	4: (*wait for answer - upload*)
		TimeStart 							:= TRUE; 						// restart timer fot timeout (for each packet)
		// expect and save packet
		IF FML_REF.RespID = FML_FPC_RESP_file_done AND FML_REF.FPCS_Packet.Control = FML_REF.FPCC_Packet.Control AND FML_REF.FPCS_Packet.BitSequenceNr = Sequence THEN
			Buffer							:= FML_REF.FPCS_Packet.Data;	// write incoming data from controller into buffer (6 Byte)
			FOR i := 0 TO 5 DO
				PtrToDataFileArray^			:= Buffer[i+1];					// write data from buffer to output (each byte separately)
				PtrToDataFileArray			:= PtrToDataFileArray + 1;
			END_FOR
			
			CountByte 						:= CountByte + udLength;		// count up the bytes
			NextSequence();       											// count sequence
			TimeStart						:= FALSE;
			Step							:= 3; 
		
		// finish upload, controller sends stopp
		ELSIF FML_REF.RespID = FML_FPC_RESP_file_done AND FML_REF.FPCS_Packet.Control = FML_FPC_FILE_TRANSFER_stop AND FML_REF.FPCS_Packet.BitSequenceNr = Sequence THEN
			TimeStart 						:= FALSE;
			IF CountByte <> Filesize OR CountByte < 100 THEN 				// check if all bytes are uploaded
				Step 			    		:= 21; 							// wrong size --> error state
				Status.Err:=TRUE; Status.Cat:=FML_parameter_transfer; Status.ID:=FML_incomplete; 
			ELSE
				Step 			    		:= 20;							// size is right, upload successful, end state		
			END_IF
						
		// error from controller, general EFPC error
		ELSIF FML_REF.RespID = FML_FPC_RESP_error THEN
			Status.Err:=TRUE; Status.Cat:=FML_parameter_transfer; Status.ID:=FML_REF.FPCS_Packet.Data[1]+1000; 
			TimeStart 						:= FALSE;
			NextSequence();     											// count sequence modul
			Step 			  				:= 23;  						// send stopp after error
			
		// error from controller - upload
		ELSIF FML_REF.FPCS_Packet.Control = FML_FPC_FILE_TRANSFER_error THEN
			Status.Err:=TRUE; Status.Cat:=FML_parameter_transfer; Status.ID:=FML_REF.FPCS_Packet.Data[1]+1000; 	// get error code from data at byte 1
			TimeStart						:= FALSE;
			NextSequence();     											// count sequence modulo
			Step							:= 23;  						// send stopp after error	
		
		ELSE 
			//timeout
			IF TimeStop THEN
				Status.Err:=TRUE; Status.Cat:=FML_parameter_transfer; Status.ID:=FML_time_out; 
				Step						:= 21;  						// send error message to controller
				TimeStart					:= FALSE;
			END_IF	
		END_IF
	
	6: (*start requirement - download*)
		FOR i := 0 TO 5 DO
			Buffer[i+1]						:= PtrToDataFileArray^;			// write data from data array (input) into buffer (each byte separately)
			PtrToDataFileArray				:= PtrToDataFileArray + 1;
		END_FOR

		IF Sequence = 0 THEN    											
			CalculateFilesize(); 											// calculate size of file as a multiple of udLength
			
			IF FileSize < 262 THEN  										// file larger than header --> error
				Step 						:= 27;
				Status.Err:=TRUE; Status.Cat:=FML_parameter_transfer; Status.ID:=FML_size_err; 
				RETURN;
			ELSIF FileSize > SizeOfFileArray THEN							// check if the array is big enough
				Step 			    		:= 27; 							// array is to small --> error state
				Status.Err:=TRUE; Status.Cat:=FML_parameter_transfer; Status.ID:=FML_volume_err;
				RETURN;
			END_IF
		END_IF	
				
		FML_REF.FPCC_Packet.Data 			:= Buffer;						// write data from buffer to controller (6 byte)	
		CountByte 							:= CountByte + udLength;
		FML_REF.FPCC_Modus					:= 4;							// modus parameter file 
		FML_REF.ReqID						:= FML_FPC_REQ_write_file; 		// download
		FML_REF.FPCC_Packet.Control			:= FML_FPC_FILE_TRANSFER_start; // start transfer
		FML_REF.FPCC_Packet.BitSequenceNr	:= Sequence;
		TimeStart 							:= TRUE;
		Step 								:= 7;

			
	7: (*wait for response from controller - download*)
		IF FML_REF.RespID = FML_FPC_RESP_file_done AND FML_REF.FPCS_Packet.Control = FML_REF.FPCC_Packet.Control AND FML_REF.FPCS_Packet.BitSequenceNr = Sequence THEN
			Sequence 						:= 1;
			Step 							:= 8;
		ELSE
			//timeout
			IF TimeStop THEN
				TimeStart 					:= FALSE;
				Step 						:= 9;
			END_IF
		END_IF

	8: (*send packet - download*)
		IF CountByte < FileSize THEN
			FOR i := 0 TO 5 DO
				Buffer[i+1]					:= PtrToDataFileArray^;			// write data from data array (input) into buffer (each byte separately)
			PtrToDataFileArray				:= PtrToDataFileArray + 1;
		END_FOR
		
		FML_REF.FPCC_Packet.Data 				:= Buffer;					// write data from buffer to controller (6 byte)
			CountByte							:= CountByte + udLength;
			FML_REF.FPCC_Packet.Control			:= FML_FPC_FILE_TRANSFER_active;
			FML_REF.FPCC_Packet.BitSequenceNr	:= Sequence;
			Step								:= 9;
				
		ELSE          //---- end of file detected -ä stop to device
			FML_REF.FPCC_Packet.Control 		:= FML_FPC_FILE_TRANSFER_stop;
			FML_REF.FPCC_Packet.BitSequenceNr	:= Sequence;
			FML_REF.FPCC_Packet.Data 			:= Buffer;
			Step								:= 9;
		END_IF
	
	9: (*wait for confirmation of receipt of controller - download*)
		// receive and process message 
		TimeStart								:= TRUE;
		IF FML_REF.RespID = FML_FPC_RESP_file_done AND FML_REF.FPCS_Packet.Control = FML_FPC_FILE_TRANSFER_active AND FML_REF.FPCS_Packet.BitSequenceNr = Sequence THEN
			NextSequence();														// count sequence modulo
			TimeStart							:= FALSE;       												
			Step								:= 8;
			
		// if stop has been sent to the controller
		ELSIF FML_REF.RespID = FML_FPC_RESP_file_done AND FML_REF.FPCS_Packet.Control = FML_FPC_FILE_TRANSFER_stop AND FML_REF.FPCS_Packet.BitSequenceNr = Sequence THEN
			IF CountByte <> Filesize OR CountByte < 100 THEN 					// check if parameterfile has been loaded
				Step 			:= 21; 											// wrong size, error step
				Status.Err:=TRUE; Status.Cat:=FML_parameter_transfer; Status.ID:=FML_incomplete;
			ELSE
				Step 			:= 20;											// right size, download successful, end state    // check if all bytes are uploaded
			END_IF
			TimeStart 			:= FALSE;
			
		// error from controller, general EFPC error
		ELSIF FML_REF.RespID = FML_FPC_RESP_error THEN
			Status.Err:=TRUE; Status.Cat:=FML_parameter_transfer; Status.ID:=FML_REF.FPCS_Packet.Data[1]+1000;	// get error code from data at byte 1
			NextSequence();       												// count sequence modulo
			Step				:= 23;
			TimeStart 			:= FALSE;
			
		// error form controller - Download
		ELSIF FML_REF.FPCS_Packet.Control = FML_FPC_FILE_TRANSFER_error THEN
			Status.Err:=TRUE; Status.Cat:=FML_parameter_transfer; Status.ID:=FML_REF.FPCS_Packet.Data[1]+1000;	// get error code from data at byte 1
      		NextSequence();       												// count sequence modulo
			IF Status.ID = FML_par_file_err THEN								// If Status.ID == 1008
				Step 			:= 27;
			ELSE
				Step 			:= 23;
			END_IF
			TimeStart 			:= FALSE;
		
		ELSE
			// timeout
			IF TimeStop THEN
				Status.Err:=TRUE; Status.Cat:=FML_parameter_transfer; Status.ID:=FML_time_out; 
				Step 			:= 21;
				TimeStart		:= FALSE;
			END_IF
		END_IF
	
	20:	(*  ==== done with no error ==== *)
		Status.Err:=FALSE; Status.Cat:=FML_no_category; Status.ID:=FML_no_error;
		Step					:= 27;      						// wait for NOT execute
	
		
	21: (*send error message to Controller*)
		NextSequence();      				 						// count sequence modulo
		FML_REF.FPCC_Modus 					:= 4;
		FML_REF.FPCC_Packet.Control 		:= 3;
		FML_REF.FPCC_Packet.BitSequenceNr  	:= Sequence;
		FML_REF.FPCC_Packet.Data 			:= Buffer;
		TimeStart							:= TRUE;
		Step 								:= 22;
			
	22: (*wait for error message from controller*)
		IF FML_REF.RespID = FML_FPC_RESP_file_done AND FML_REF.FPCS_Packet.Control = FML_FPC_FILE_TRANSFER_error THEN
			NextSequence();       									// count sequence modulo
			TimeStart						:= FALSE;
			Step 							:= 23;
		ELSE
			IF TimeStop THEN
				Status.Err:=TRUE; Status.Cat:=FML_parameter_transfer; Status.ID:=FML_time_out;
				TimeStart 					:= FALSE;
				Step 						:= 23;
			END_IF
		END_IF
		
	23: (*send STOPP after error*)	
		FML_REF.FPCC_Packet.Control 		:= 2; 					// after error STOPP is sending to Controller
		FML_REF.FPCC_Packet.BitSequenceNr 	:= Sequence;
		FML_REF.FPCC_Packet.Data 			:= Buffer;
		TimeStart 							:= TRUE;
		Step 								:= 24;		
		
	24: (*query wheater stop was confirmed by controller*)
		IF (FML_REF.RespID = FML_FPC_RESP_file_done AND FML_REF.FPCS_Packet.Control = 2) OR  FML_REF.RespID = 7 THEN
			Step 							:= 27;
			TimeStart 						:= FALSE;
		ELSIF FML_REF.RespID = FML_FPC_RESP_file_done AND FML_REF.FPCS_Packet.Control = 3 AND SendRepeat < 4 THEN
			Status.ID						:= FML_REF.FPCS_Packet.Data[1]+1000;			// get error code from data at byte 1
			IF Status.ID <> 1000 THEN
				Status.Err					:= TRUE;
				Status.Cat					:= FML_parameter_transfer;
			END_IF
			
			Sequence 						:= Sequence + 1;
			SendRepeat 						:= SendRepeat + 1;
			TimeStart 						:= FALSE;
			Step 							:= 23;
		ELSE
			// timeout
			IF TimeStop THEN
				Status.Err:=TRUE; Status.Cat:=FML_parameter_transfer; Status.ID:=FML_time_out;
				TimeStart 					:= FALSE;
				Step 						:= 27;
			END_IF
		END_IF
		
  
  27: (*idle - wait for execute = false*)
		vis_upload 							:= FALSE;
		vis_download 						:= FALSE;
		Done								:= TRUE;
		Step								:= 30;
    		
  30: (*do nothing - wait for NOT execute*)
    	;
  
END_CASE

Status.Msg				:= GetStatusMessage(Status);
Error					:= Status.Err;

(* ===== end of function block ============================= *)

ACTION CalculateFilesize:
(* -----------------------------------------------------
   This action calculates the file size as a couple of 6 
   from the first 2 bytes of the buffer
   ----------------------------------------------------- *)

 	FileSize	:= DWORD_TO_DINT( SHL(BYTE_TO_DWORD(pbyBuffer^[2]),8) OR pbyBuffer^[1]); 	// length of data field
	FileSize	:= (Filesize + 2 * udLength -1) / udLength ; 								// +6: size of parameter file at first position, +5 und /6 for rounding up 
	FileSize	:= FileSize * udLength; 													// bytesize is being computed out of number of packages
END_ACTION

ACTION NextSequence:
(* -----------------------------------------------------
   This action increments the Sequence counter modulo 32. 
   It is used at 8 points in CMMO_ST_PRM_FILE
   ----------------------------------------------------- *)
	IF Sequence = 31 THEN
		Sequence 	:= 0;
	ELSE
		Sequence 	:= Sequence + 1;
	END_IF
END_ACTION

END_FUNCTION_BLOCK

// Blocks/Parameterize/FPC_DIRMP
(* ============================================================================
   FESTO AG & Co. KG, Esslingen - Copyright 2015. All rights reserved.                       
 ------------------------------------------------------------------------------
 Functionblock:  PRM_DIRMP  
 Description:    function block to pass dynamic parameter values for direct-mode-positioncontrol
 Version:        V3.5.7.21        
 Composer:       bejk
 Last update:    13.11.2017                                                                           
------------------------------------------------------------------------------- *)
{library private}
(* -----------------------------------------------------------------------------
Date        Name            	Activity                                                                              
11.03.2009  Benjamin Kilgus 	created
            Rudolf Schenke  	PNU array created 
09.02.2015  Rudolf Schenke  	Implement 16-bit mode with hide preset 
22.06.2015	Christian Hammer	adaptation to use this FB for all drives
04.09.2015  Christian Hammer	error handling (deleted RETVAL, created Status)
13.11.2017	Christian Hammer	added blockade of FB for SFC-DC and MTR-DCI controller
=============================================================================== *)
{library public}

(* use this function block only with the function blocks FML_Read and FML_Write *)

FUNCTION_BLOCK FPC_DIRMP

VAR_IN_OUT
	FML_REF					: DT_FML_REF;		// structure of the parameter to control and parametrize the motorcontroller
END_VAR

VAR_INPUT
	Execute             	: BOOL;				// perfrom data exchange
	Write               	: BOOL;				// read or write the parameter	(1=write/0=read)
	Velocity            	: DINT;				// base velocity directmode positioning
	Acceleration			: DINT; 			// acceleration directmode positioning
 	Deceleration        	: DINT; 			// deceleration directmode positioning
END_VAR

VAR_OUTPUT	
	Done                	: BOOL;				// transmission done
	Error					: BOOL; 			// transmission fault
	Status					: DT_FML_STATUS;	// structure with the status information of the function block and FPC
	ActVelocity         	: DINT;  			// base velocity directmode positioning
	ActAcceleration     	: DINT;  			// acceleration directmode positioning
	ActDeceleration     	: DINT;  			// deceleration directmode positioning
END_VAR

{library private}
VAR
	bInit           		: BOOL	:=FALSE;										// status of inizialisation of the FB
	lMemberID   			: INT;													// local member ID of the FB													
	Param       			: ARRAY [1..maxParamCount] OF DT_FML_PRM_DESCRIPTION;	// parameter to write in motorcontroller
	listPNU    				: ARRAY [1..maxParamCount] OF INT := [540,541,542];		// PNUs for the parameter 
	Step        			: INT:= 0; 												// actual step number 
	ixPar       			: INT:= 1;  											// index for the array

	TONInst					: TON;													// timer instance to monitor a timeout of the function block
	TimeStart				: BOOL;													// variable to start the timer instance
	TimeoutTime				: TIME := T#3S;											// timeout time 	
END_VAR

VAR CONSTANT
	maxParamCount			: INT := 3;												// max number of the parameter 
END_VAR

{library public}

(* ====== initial block routine ===================================== *)
(* ----- get MemberID for this function block ------------------------*)
IF NOT bInit THEN
	FML_REF.MemberIDmax		:= FML_REF.MemberIDmax +1;
	lMemberID				:= FML_REF.MemberIDmax;
	bInit					:= TRUE;
	Status.Err:=FALSE; Status.Cat:=FML_function_block; Status.ID:=FML_init_active;
END_IF


(* ====== supervision of timeout ==================================== *)
(* ----- timer to monitor a timeout of the function block ------------*)
TONInst(IN := TimeStart, PT := TimeoutTime);
IF TONInst.Q THEN
	Status.Err:=TRUE; Status.Cat:=FML_function_block; Status.ID:=FML_fb_timeout;
	Done					:= TRUE;
	Step					:= 30;
END_IF

// this function block is not usable with SFC-DC and MTR-DCI
IF Execute 
	AND	((FML_REF.DeviceType = SFC_DC)
	OR (FML_REF.DeviceType = MTR_DCI)) THEN
		Done				:= TRUE;
		Status.Err:=TRUE; Status.Cat:=FML_function_block; Status.ID:=FML_wrong_device;
		Step				:= 100;
END_IF

IF Param[1].PNU = 0 THEN
  FOR ixPar:=1 TO maxParamCount DO
    Param[ixPar].PNU 		:= listPNU[ixPar]; 			// fill in the PNU
    Param[ixPar].SUBINDEX 	:= 1;         				// fill in a fix subindex
	END_FOR
    // 1 =  540.1: Paramter Direktbetrieb Basisgeschwindigkeit directmode positioning
    // 2 =  541.1: Paramter Beschleunigung directmode positioning
    // 3 =  542.1: Paramter Verzögerung directmode positioning
END_IF;

(* ===== logic part ================================================= *)
IF NOT Execute AND (Step <> 0) THEN   					// aborting FB
	FML_REF.MemberID		:= 0;
	FML_REF.ReqID        	:= FML_FPC_REQ_none;
	FML_REF.PNU       		:= 0;
	FML_REF.Subindex   		:= 0;
	FML_REF.Value			:= 0;
	ActVelocity				:= 0;
	ActAcceleration			:= 0;
	ActDeceleration			:= 0;
 	Step                    := 0;
END_IF

CASE Step OF
  0:(* *)
  Done						:= FALSE;
  TimeStart					:= FALSE;
  Status.Err:=FALSE; Status.Cat:=FML_no_category; Status.ID:=FML_no_error;

	IF (FML_REF.MemberID = 0) AND Execute THEN 	
		Status.Err:=FALSE; Status.Cat:=FML_function_block; Status.ID:=FML_fb_busy;
		
		IF (FML_REF.DeviceType = CMMP_AS) 
		OR (FML_REF.DeviceType = CMMS_AS) 
		OR (FML_REF.DeviceType = CMMS_ST)
		OR (FML_REF.DeviceType = CMMD_AS) THEN					(* CMMP-AS or CMMS_AS or CMMS_ST or CMMD_AS *)	
			FML_REF.FPCC_Modus 	:= E_FML_FPC_MODUS.FML_FPC_MODUS_PNU_11BIT;
		ELSE 												(*******EMCA-EC or CMMO-ST*******)	
			FML_REF.FPCC_Modus 	:= E_FML_FPC_MODUS.FML_FPC_MODUS_PNU_16BIT;
		END_IF
    	FML_REF.MemberID		:= lMemberID;
		FML_REF.ReqID			:= FML_FPC_REQ_none;
		FML_REF.PNU				:= 0;
		FML_REF.Subindex		:= 0;
		FML_REF.Value			:= 0;
		ixPar					:= 1;  						// set to 1st array element
		(* writing *)
		IF Write THEN
			Param[1].Value		:= Velocity;
			Param[2].Value		:= Acceleration;
			Param[3].Value		:= Deceleration;
			Step				:= 10;
		(* reading *)
		ELSE
			Step				:= 20;
		END_IF
	ELSIF (FML_REF.MemberID <> lMemberId) AND Execute THEN
		Status.Err:=FALSE; Status.Cat:=FML_function_block; Status.ID:=FML_other_fb_active;
	END_IF

  10:(* writing parameter[ixPar] *)
  	TimeStart					:= TRUE;
	IF NOT FML_REF.Done THEN
		TimeStart				:= FALSE;  
		FML_REF.ReqID			:= FML_FPC_REQ_write_array_dword;
		FML_REF.PNU				:= Param[ixPar].PNU;
		FML_REF.Subindex		:= Param[ixPar].SUBINDEX;
		FML_REF.Value			:= Param[ixPar].VALUE;
		Step					:= 11;
	END_IF

  11:(* *)
  	TimeStart					:= TRUE;
	IF FML_REF.Done AND NOT FML_REF.Err THEN
		TimeStart				:= FALSE;
		FML_REF.ReqID			:= FML_FPC_REQ_none;
		ixPar					:= ixPar +1;
		Step					:= 10;
		IF ixPar > maxParamCount THEN
		  	Done					:= TRUE;
		  	ActVelocity			:= Param[1].VALUE;
			ActAcceleration		:= Param[2].VALUE;
			ActDeceleration		:= Param[3].VALUE;
		  	Status.Err:=FALSE; Status.Cat:=FML_no_category; Status.ID:=FML_no_error;
		  	Step				:= 30;
		END_IF
	ELSIF FML_REF.Done AND FML_REF.Err THEN
		TimeStart				:= FALSE; 
		Done					:= TRUE;
		Status.Err:=TRUE; Status.Cat:=FML_parameter_transfer; Status.ID:=FML_REF.ActValue;
		Step					:= 30;
	END_IF

  20: (* reading *)
  	TimeStart					:= TRUE;
	IF NOT FML_REF.Done THEN
		TimeStart				:= FALSE;
		FML_REF.ReqID			:= FML_FPC_REQ_read_array;
 		FML_REF.PNU				:= Param[ixPar].PNU;
 		FML_REF.Subindex		:= Param[ixPar].SUBINDEX;
 		Step					:= 21;
	END_IF

  21:(* set ouput variables*)
  	TimeStart					:= TRUE;
	IF FML_REF.Done AND NOT FML_REF.Err THEN
		TimeStart				:= FALSE;  
		FML_REF.ReqID			:= FML_FPC_REQ_none;
		Param[ixPar].Value		:= FML_REF.ActValue;
		ixPar					:= ixPar +1;
		Step					:= 20;
		IF ixPar > maxParamCount THEN
			ActVelocity			:= Param[1].VALUE;
			ActAcceleration		:= Param[2].VALUE;
			ActDeceleration		:= Param[3].VALUE;
			Done				:= TRUE;
			Status.Err:=FALSE; Status.Cat:=FML_no_category; Status.ID:=FML_no_error;
			Step				:= 30;
		END_IF
	ELSIF FML_REF.Done AND FML_REF.Err THEN
		TimeStart				:= FALSE;  
		Done					:= TRUE;
		Status.Err:=TRUE; Status.Cat:=FML_parameter_transfer; Status.ID:=FML_REF.ActValue;
		Step					:= 30;
	END_IF

  30: (* done - do nothing *)
	  ;
	  
END_CASE;

Status.Msg				:= GetStatusMessage(Status);
Error					:= Status.Err;

(* ===== end of function block ============================= *)

END_FUNCTION_BLOCK

// VISU/VIS_FPC_PNU
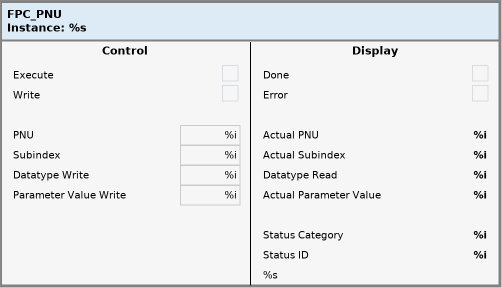
VISUALIZATION VIS_FPC_PNU  // 502x288
VAR_INPUT
	{attribute 'parameterstringof' := 'm_Input_INST'}
	m_Input_INST_Str 	: STRING;
END_VAR
VAR_IN_OUT
	m_Input_INST 		: FPC_PNU;
END_VAR
    Rectangle (0,1 500x285)
    Rectangle (0,1 500x40), "FPC_PNU Instance: %s", text variable: m_Input_INST_Str
    Rectangle (260,265 240x20), "%s", text variable: m_Input_INST.Status.Msg
    Rectangle (180,125 60x20), "%i", text variable: m_Input_INST.PNU
        OnMouseDown: write the text variable via Edit
    Rectangle (180,165 60x20), "%i", text variable: m_Input_INST.DatatypeWR
        OnMouseDown: write the text variable via Edit
    Rectangle (430,125 60x20), "%i", text variable: m_Input_INST.ActPNU
    Label (10,65 120x20), "Execute"
    Label (10,85 120x20), "Write"
    RoundedRectangle (222,65 16x16), colour toggle: m_Input_INST.Execute
        toggle m_Input_INST.Execute
    RoundedRectangle (222,85 16x16), colour toggle: m_Input_INST.Write
        toggle m_Input_INST.Write
    Label (10,125 120x20), "PNU"
    Label (10,165 120x20), "Datatype Write"
    Label (260,65 120x20), "Done"
    Label (260,85 120x20), "Error"
    RoundedRectangle (472,65 16x16), colour toggle: m_Input_INST.Done
    RoundedRectangle (472,85 16x16), colour toggle: m_Input_INST.Error
    Label (260,125 128x20), "Actual PNU"
    Label (0,41 250x20), "Control"
    Label (250,41 250x20), "Display"
    Line (250,42) (250,285)
    Rectangle (430,165 60x20), "%i", text variable: m_Input_INST.DatatypeRD
    Label (260,165 128x20), "Datatype Read"
    Rectangle (180,145 60x20), "%i", text variable: m_Input_INST.Subindex
        OnMouseDown: write the text variable via Edit
    Rectangle (430,145 60x20), "%i", text variable: m_Input_INST.ActSubindex
    Label (10,145 120x20), "Subindex"
    Label (260,145 128x20), "Actual Subindex"
    Rectangle (430,225 60x20), "%i", text variable: m_Input_INST.Status.Cat
    Label (260,225 128x20), "Status Category"
    Rectangle (430,245 60x20), "%i", text variable: m_Input_INST.Status.ID
    Label (260,245 128x20), "Status ID"
    Rectangle (180,185 60x20), "%i", text variable: m_Input_INST.Value
        OnMouseDown: write the text variable via Edit
    Label (10,185 120x20), "Parameter Value Write"
    Rectangle (430,185 60x20), "%i", text variable: m_Input_INST.ActValue
    Label (260,185 128x20), "Actual Parameter Value"
END_VISUALIZATION

// VISU/VIS_FPC_DIAG_BUFFER
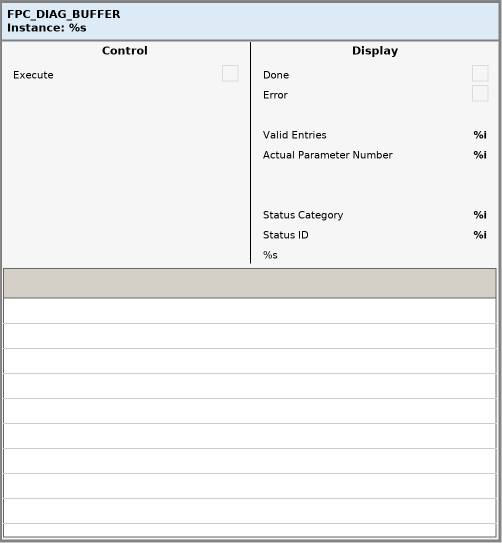
VISUALIZATION VIS_FPC_DIAG_BUFFER  // 502x543
VAR_INPUT
	{attribute 'parameterstringof' := 'm_Input_INST'}
	m_Input_INST_Str 	: STRING;
END_VAR
VAR_IN_OUT
	m_Input_INST 		: FPC_DIAG_BUFFER;
END_VAR
    Rectangle (0,1 500x540)
    Rectangle (0,1 500x40), "FPC_DIAG_BUFFER Instance: %s", text variable: m_Input_INST_Str
    Rectangle (260,245 240x20), "%s", text variable: m_Input_INST.Status.Msg
    Rectangle (430,145 60x20), "%i", text variable: m_Input_INST.ParamNo
    Label (10,65 120x20), "Execute"
    RoundedRectangle (222,65 16x16), colour toggle: m_Input_INST.Execute
        toggle m_Input_INST.Execute
    Label (260,65 120x20), "Done"
    Label (260,85 120x20), "Error"
    RoundedRectangle (472,65 16x16), colour toggle: m_Input_INST.Done
    RoundedRectangle (472,85 16x16), colour toggle: m_Input_INST.Error
    Label (260,145 140x20), "Actual Parameter Number"
    Label (0,41 250x20), "Control"
    Label (250,41 250x20), "Display"
    Line (250,42) (250,263)
    Rectangle (430,205 60x20), "%i", text variable: m_Input_INST.Status.Cat
    Label (260,205 128x20), "Status Category"
    Rectangle (430,225 60x20), "%i", text variable: m_Input_INST.Status.ID
    Label (260,225 128x20), "Status ID"
    Rectangle (430,125 60x20), "%i", text variable: m_Input_INST.ValidEntries
    Label (260,125 140x20), "Valid Entries"
    Table (3,268 493x269), data array: m_Input_INST.astVisu
        p3854506369: m_Input_INST.astVisu[INDEX].sEvent
        p1892666644: m_Input_INST.astVisu[INDEX].sStamp
        p338671338: m_Input_INST.astVisu[INDEX].sFault
        p2170511999: m_Input_INST.astVisu[INDEX].sText
        p511219082: TimeStamp
        p1755163831: Message #
        p4092479075: Message Description
END_VISUALIZATION

// VISU/VIS_FPC_DIRMP
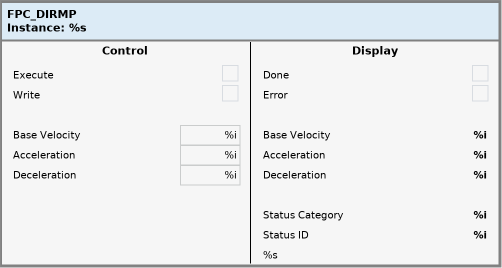
VISUALIZATION VIS_FPC_DIRMP  // 502x268
VAR_INPUT
	{attribute 'parameterstringof' := 'm_Input_INST'}
	m_Input_INST_Str 	: STRING;
END_VAR
VAR_IN_OUT
	m_Input_INST 		: FPC_DIRMP;
END_VAR
    Rectangle (0,1 500x265)
    Rectangle (0,1 500x40), "FPC_DIRMP Instance: %s", text variable: m_Input_INST_Str
    Rectangle (260,245 240x20), "%s", text variable: m_Input_INST.Status.Msg
    Rectangle (180,125 60x20), "%i", text variable: m_Input_INST.Velocity
        OnMouseDown: write the text variable via Edit
    Rectangle (180,165 60x20), "%i", text variable: m_Input_INST.Deceleration
        OnMouseDown: write the text variable via Edit
    Rectangle (430,125 60x20), "%i", text variable: m_Input_INST.ActVelocity
    Label (10,65 120x20), "Execute"
    Label (10,85 120x20), "Write"
    RoundedRectangle (222,65 16x16), colour toggle: m_Input_INST.Execute
        toggle m_Input_INST.Execute
    RoundedRectangle (222,85 16x16), colour toggle: m_Input_INST.Write
        toggle m_Input_INST.Write
    Label (10,125 120x20), "Base Velocity"
    Label (10,165 120x20), "Deceleration"
    Label (260,65 120x20), "Done"
    Label (260,85 120x20), "Error"
    RoundedRectangle (472,65 16x16), colour toggle: m_Input_INST.Done
    RoundedRectangle (472,85 16x16), colour toggle: m_Input_INST.Error
    Label (260,125 128x20), "Base Velocity"
    Label (0,41 250x20), "Control"
    Label (250,41 250x20), "Display"
    Line (250,42) (250,263)
    Rectangle (430,165 60x20), "%i", text variable: m_Input_INST.ActDeceleration
    Label (260,165 128x20), "Deceleration"
    Rectangle (180,145 60x20), "%i", text variable: m_Input_INST.Acceleration
        OnMouseDown: write the text variable via Edit
    Rectangle (430,145 60x20), "%i", text variable: m_Input_INST.ActAcceleration
    Label (10,145 120x20), "Acceleration"
    Label (260,145 128x20), "Acceleration"
    Rectangle (430,205 60x20), "%i", text variable: m_Input_INST.Status.Cat
    Label (260,205 128x20), "Status Category"
    Rectangle (430,225 60x20), "%i", text variable: m_Input_INST.Status.ID
    Label (260,225 128x20), "Status ID"
END_VISUALIZATION

// VISU/VIS_FPC_DATA_OBJECT
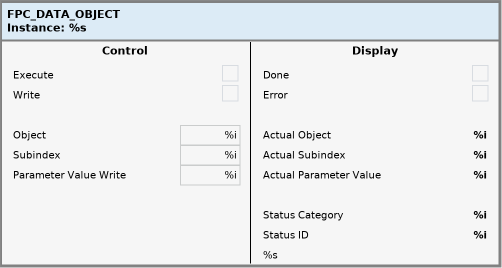
VISUALIZATION VIS_FPC_DATA_OBJECT  // 502x268
VAR_INPUT
	{attribute 'parameterstringof' := 'm_Input_INST'}
	m_Input_INST_Str	: STRING;
END_VAR
VAR_IN_OUT
	m_Input_INST 		: FPC_DATA_OBJECT;
END_VAR
    Rectangle (0,1 500x265)
    Rectangle (0,1 500x40), "FPC_DATA_OBJECT Instance: %s", text variable: m_Input_INST_Str
    Rectangle (260,245 240x20), "%s", text variable: m_Input_INST.Status.Msg
    Rectangle (180,125 60x20), "%i", text variable: m_Input_INST.Object
        OnMouseDown: write the text variable via Edit
    Rectangle (180,165 60x20), "%i", text variable: m_Input_INST.Value
        OnMouseDown: write the text variable via Edit
    Rectangle (430,125 60x20), "%i", text variable: m_Input_INST.ActObject
    Label (10,65 120x20), "Execute"
    Label (10,85 120x20), "Write"
    RoundedRectangle (222,65 16x16), colour toggle: m_Input_INST.Execute
        toggle m_Input_INST.Execute
    RoundedRectangle (222,85 16x16), colour toggle: m_Input_INST.Write
        toggle m_Input_INST.Write
    Label (10,125 120x20), "Object"
    Label (10,165 120x20), "Parameter Value Write"
    Label (260,65 120x20), "Done"
    Label (260,85 120x20), "Error"
    RoundedRectangle (472,65 16x16), colour toggle: m_Input_INST.Done
    RoundedRectangle (472,85 16x16), colour toggle: m_Input_INST.Error
    Label (260,125 128x20), "Actual Object"
    Label (0,41 250x20), "Control"
    Label (250,41 250x20), "Display"
    Line (250,42) (250,263)
    Rectangle (430,165 60x20), "%i", text variable: m_Input_INST.ActValue
    Label (260,165 128x20), "Actual Parameter Value"
    Rectangle (180,145 60x20), "%i", text variable: m_Input_INST.Subindex
        OnMouseDown: write the text variable via Edit
    Rectangle (430,145 60x20), "%i", text variable: m_Input_INST.ActSubindex
    Label (10,145 120x20), "Subindex"
    Label (260,145 128x20), "Actual Subindex"
    Rectangle (430,205 60x20), "%i", text variable: m_Input_INST.Status.Cat
    Label (260,205 128x20), "Status Category"
    Rectangle (430,225 60x20), "%i", text variable: m_Input_INST.Status.ID
    Label (260,225 128x20), "Status ID"
END_VISUALIZATION

// VISU/VIS_FHPP_CTRL
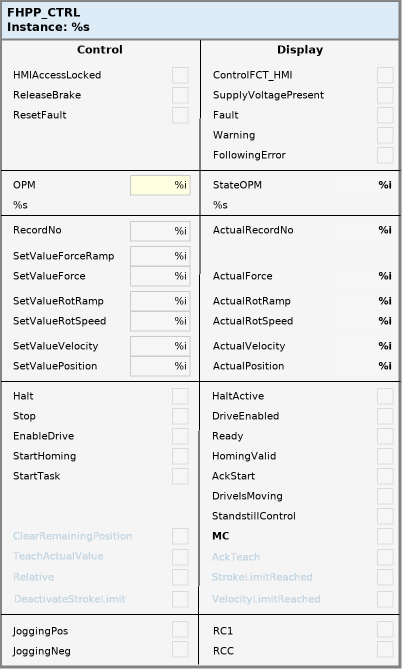
VISUALIZATION VIS_FHPP_CTRL  // 402x669
VAR_INPUT
	{attribute 'parameterstringof' := 'm_Input_INST'}
	m_Input_INST_Str 	: STRING;
END_VAR
VAR_IN_OUT
	m_Input_INST 		: FHPP_CTRL;
END_VAR
    Rectangle (0,1 400x666)
    Rectangle (0,0 400x40), "FHPP_CTRL Instance: %s", text variable: m_Input_INST_Str
    Rectangle (10,195 180x20), "%s", text variable: m_Input_INST.OPMString
    Rectangle (130,266 60x20), "%i", text variable: m_Input_INST.SetValueForce, colour toggle: (m_Input_INST.OPM) = 5
        OnMouseDown: write the text variable via Edit
    Rectangle (330,175 65x20), "%i", text variable: m_Input_INST.StateOPM
    Rectangle (130,336 60x20), "%i", tooltip "permissible range of value is 0 to 100", text variable: m_Input_INST.SetValueVelocity, colour toggle: (m_Input_INST.OPM= 1) or ((m_Input_INST.OPM =5) AND (m_Input_INST.tempVisuMode =2))
        OnMouseDown: write the text variable via Edit
    Rectangle (335,336 60x20), "%i", text variable: m_Input_INST.ActualVelocity, colour toggle: (m_Input_INST.StateOPM) = 1
    Rectangle (130,291 60x20), "%i", tooltip "permissible range of value is 0 to 100", text variable: m_Input_INST.SetValueRotRamp, colour toggle: m_Input_INST.OPM = 9
        OnMouseDown: write the text variable via Edit
    Rectangle (335,291 60x20), "%i", text variable: m_Input_INST.ActualRotRamp, colour toggle: (m_Input_INST.StateOPM) = 9
    Rectangle (130,311 60x20), "%i", text variable: m_Input_INST.SetValueRotSpeed, colour toggle: (m_Input_INST.OPM) = 9
        OnMouseDown: write the text variable via Edit
    Rectangle (335,311 60x20), "%i", text variable: m_Input_INST.ActualRotSpeed, colour toggle: (m_Input_INST.StateOPM) = 9
    Rectangle (130,356 60x20), "%i", text variable: m_Input_INST.SetValuePosition, colour toggle: (m_Input_INST.OPM) = 1
        OnMouseDown: write the text variable via Edit
    Rectangle (335,356 60x20), "%i", text variable: m_Input_INST.ActualPosition, colour toggle: (m_Input_INST.StateOPM = 1) or (m_Input_INST.StateOPM = 5) or (m_Input_INST.StateOPM = 0)
    Rectangle (210,195 180x20), "%s", text variable: m_Input_INST.StateOPMString
    Rectangle (335,266 60x20), "%i", text variable: m_Input_INST.ActualForce, colour toggle: (m_Input_INST.StateOPM) = 5
    Rectangle (335,220 60x20), "%i", text variable: m_Input_INST.ActualRecordNo, colour toggle: (m_Input_INST.StateOPM) = 0
    RoundedRectangle (377,428 16x16), colour toggle: m_Input_Inst.Ready
    RoundedRectangle (172,428 16x16), colour toggle: m_Input_Inst.EnableDrive
        toggle m_Input_Inst.EnableDrive
    RoundedRectangle (172,388 16x16), colour toggle: m_Input_Inst.Halt
        toggle m_Input_Inst.Halt
    RoundedRectangle (172,408 16x16), colour toggle: m_Input_Inst.Stop
        toggle m_Input_Inst.Stop
    RoundedRectangle (377,388 16x16), colour toggle: m_Input_Inst.HaltActive
    RoundedRectangle (377,408 16x16), colour toggle: m_Input_Inst.DriveEnabled
    RoundedRectangle (172,448 16x16), colour toggle: m_Input_Inst.StartHoming
        toggle m_Input_Inst.StartHoming
    RoundedRectangle (172,468 16x16), colour toggle: m_Input_Inst.StartTask
        toggle m_Input_Inst.StartTask
    RoundedRectangle (172,549 16x16), colour toggle: m_Input_Inst.TeachActualValue
        toggle m_Input_Inst.TeachActualValue
    RoundedRectangle (172,528 16x16), colour toggle: m_Input_Inst.ClearRemainingPosition
        toggle m_Input_Inst.ClearRemainingPosition
    RoundedRectangle (172,569 16x16), colour toggle: m_Input_Inst.Relative
        toggle m_Input_INST.Relative
    RoundedRectangle (377,448 16x16), colour toggle: m_Input_Inst.HomingValid
    RoundedRectangle (377,468 16x16), colour toggle: m_Input_Inst.AckStart
    RoundedRectangle (377,488 16x16), colour toggle: m_Input_Inst.DriveIsMoving
    RoundedRectangle (377,508 16x16), colour toggle: m_Input_Inst.StandstillControl
    RoundedRectangle (377,528 16x16), colour toggle: m_Input_Inst.MC
    RoundedRectangle (377,621 16x16), colour toggle: m_Input_Inst.RC1
    RoundedRectangle (377,641 16x16), colour toggle: m_Input_Inst.RCC
    Label (10,65 140x20), "HMIAccessLocked"
    Label (10,85 140x20), "ReleaseBrake"
    Label (10,105 140x20), "ResetFault"
    RoundedRectangle (172,621 16x16), colour toggle: m_Input_Inst.JoggingPos
        toggle m_Input_Inst.JoggingPos
    RoundedRectangle (172,641 16x16), colour toggle: m_Input_Inst.JoggingNeg
        toggle m_Input_Inst.JoggingNeg
    RoundedRectangle (172,67 16x16), colour toggle: m_Input_Inst.HMIAccessLocked
        toggle m_Input_Inst.HMIAccessLocked
    RoundedRectangle (172,87 16x16), colour toggle: m_Input_Inst.Brake
        toggle m_Input_Inst.Brake
    RoundedRectangle (172,107 16x16), colour toggle: m_Input_Inst.ResetFault
        toggle m_Input_Inst.ResetFault
    RoundedRectangle (377,67 16x16), colour toggle: m_Input_Inst.ControlFCT_HMI
    RoundedRectangle (377,87 16x16), colour toggle: m_Input_Inst.SupplyVoltagePresent
    RoundedRectangle (377,107 16x16), colour toggle: m_Input_Inst.Fault
    RoundedRectangle (377,127 16x16), colour toggle: m_Input_Inst.Warning
    RoundedRectangle (377,147 16x16), colour toggle: m_Input_Inst.FollowingError
    Label (210,65 120x20), "ControlFCT_HMI"
    Label (210,85 120x20), "SupplyVoltagePresent"
    Label (210,105 120x20), "Fault"
    Label (210,125 120x20), "Warning"
    Label (210,145 120x20), "FollowingError"
    Label (210,175 120x20), "StateOPM"
    Label (10,175 120x20), "OPM"
    Label (10,220 120x20), "RecordNo"
    Label (10,266 120x20), "SetValueForce"
    Label (10,291 120x20), "SetValueRotRamp"
    Label (10,311 120x20), "SetValueRotSpeed"
    Label (10,336 120x20), "SetValueVelocity"
    Label (10,356 120x20), "SetValuePosition"
    Label (10,386 120x20), "Halt"
    Label (10,406 120x20), "Stop"
    Label (10,426 120x20), "EnableDrive"
    Label (10,446 120x20), "StartHoming"
    Label (200,40 200x20), "Display"
    Label (0,40 200x20), "Control"
    Line (-1,614) (399,614)
    Line (200,40) (198,664)
    Line (0,381) (400,381)
    Line (0,215) (400,215)
    Line (0,170) (400,170)
    Label (210,220 120x20), "ActualRecordNo"
    Label (210,266 120x20), "ActualForce"
    Label (210,291 120x20), "ActualRotRamp"
    Label (210,311 120x20), "ActualRotSpeed"
    Label (210,336 120x20), "ActualVelocity"
    Label (210,356 120x20), "ActualPosition"
    Label (209,386 120x20), "HaltActive"
    Label (209,406 120x20), "DriveEnabled"
    Label (209,426 120x20), "Ready"
    Label (209,446 120x20), "HomingValid"
    Label (209,466 120x20), "AckStart"
    Label (209,486 120x20), "DriveIsMoving"
    Label (209,506 120x20), "StandstillControl"
    Label (209,526 120x20), "MC"
    Label (210,641 120x20), "RCC"
    Label (210,621 120x20), "RC1"
    Label (10,466 120x20), "StartTask"
    Label (10,621 130x20), "JoggingPos"
    Label (10,641 130x20), "JoggingNeg"
    Rectangle (130,221 60x20), "%i", text variable: m_Input_INST.RecordNo, colour toggle: (m_Input_INST.OPM) = 0
        OnMouseDown: write the text variable via Edit
    RoundedRectangle (172,591 16x16), colour toggle: m_Input_Inst.DeactivateStrokeLimit
        toggle m_Input_Inst.DeactivateStrokeLimit
    Rectangle (130,175 60x20), "%i", tooltip "0 = Record mode 1 = Direct position control 5 = Direct torque control 9 = Direct velocity control", text variable: m_Input_INST.OPM
        OnMouseDown: write the text variable via Edit
    Group (11,589 130x20)
        Label (0,0 130x20), "DeactivateStrokeLimit", invisible if: (m_Input_INST.OPM <> 5) and (m_Input_INST.OPM <> 9)
        Label (0,0 130x20), "DeactivateStrokeLimit", invisible if: (m_Input_INST.OPM = 5) or (m_Input_INST.OPM = 9)
    Group (10,546 120x20)
        Label (0,0 120x20), "TeachActualValue", invisible if: m_Input_INST.OPM <> 0
        Label (0,0 120x20), "TeachActualValue", invisible if: m_Input_INST.OPM = 0
    Group (10,567 120x20)
        Label (0,0 120x20), "Relative", invisible if: m_Input_INST.OPM <> 1
        Label (0,0 120x20), "Relative", invisible if: m_Input_INST.OPM = 1
    Group (10,526 130x20)
        Label (0,0 130x20), "ClearRemainingPosition", invisible if: (m_Input_INST.OPM <> 1) and (m_Input_INST.OPM <> 0)
        Label (0,0 130x20), "ClearRemainingPosition", invisible if: (m_Input_INST.OPM = 1) or (m_Input_INST.OPM = 0)
    RoundedRectangle (377,549 16x16), colour toggle: m_Input_Inst.AckTeach
    Group (209,547 120x20)
        Label (0,0 120x20), "AckTeach", invisible if: m_Input_INST.OPM <> 0
        Label (0,0 120x20), "AckTeach", invisible if: m_Input_INST.OPM = 0
    RoundedRectangle (377,591 16x16), colour toggle: m_Input_Inst.VelocityLimitReached
    Group (209,589 120x20)
        Label (0,0 120x20), "VelocityLimitReached", invisible if: (m_Input_INST.OPM <> 5) and (m_Input_INST.OPM <> 9)
        Label (0,0 120x20), "VelocityLimitReached", invisible if: (m_Input_INST.OPM = 5) or (m_Input_INST.OPM = 9)
    RoundedRectangle (377,569 16x16), colour toggle: m_Input_Inst.StrokeLimitReached
    Group (209,567 120x20)
        Label (0,0 120x20), "StrokeLimitReached", invisible if: (m_Input_INST.OPM <> 9) and (m_Input_INST.OPM <> 5)
        Label (0,0 120x20), "StrokeLimitReached", invisible if: (m_Input_INST.OPM = 5) or (m_Input_INST.OPM = 9)
    Rectangle (130,246 60x20), "%i", tooltip "permissible range of value is 0 to 100", text variable: m_Input_INST.SetValueForceRamp, colour toggle: (m_Input_INST.OPM = 5) AND (m_Input_INST.tempVisuMode =1)
        OnMouseDown: write the text variable via Edit
    Label (10,246 120x20), "SetValueForceRamp"
END_VISUALIZATION

// VISU/VIS_FPC_DIAG
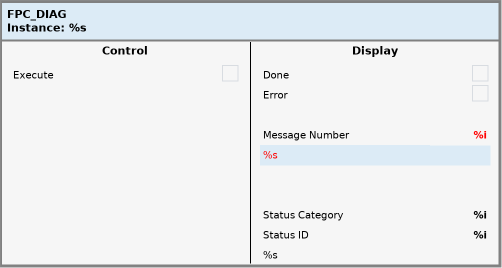
VISUALIZATION VIS_FPC_DIAG  // 502x268
VAR_INPUT
	{attribute 'parameterstringof' := 'm_Input_INST'}
	m_Input_INST_Str 	: STRING;
END_VAR
VAR_IN_OUT
	m_Input_INST 		: FPC_DIAG;
END_VAR
    Rectangle (0,1 500x265)
    Rectangle (0,1 500x40), "FPC_DIAG Instance: %s", text variable: m_Input_INST_Str
    Rectangle (260,245 240x20), "%s", text variable: m_Input_INST.Status.Msg
    Label (10,65 120x20), "Execute"
    RoundedRectangle (222,65 16x16), colour toggle: m_Input_INST.Execute
        toggle m_Input_INST.Execute
    Label (260,65 120x20), "Done"
    Label (260,85 120x20), "Error"
    RoundedRectangle (472,65 16x16), colour toggle: m_Input_INST.Done
    RoundedRectangle (472,85 16x16), colour toggle: m_Input_INST.Error
    Label (260,125 128x20), "Message Number"
    Label (0,41 250x20), "Control"
    Label (250,41 250x20), "Display"
    Line (250,42) (250,263)
    Rectangle (430,205 60x20), "%i", text variable: m_Input_INST.Status.Cat
    Label (260,205 128x20), "Status Category"
    Rectangle (430,225 60x20), "%i", text variable: m_Input_INST.Status.ID
    Label (260,225 128x20), "Status ID"
    Rectangle (260,145 230x20), "%s", text variable: m_Input_INST.MessageDescription
    Rectangle (430,125 60x20), "%i", text variable: m_Input_INST.MessageNumber
END_VISUALIZATION

// VISU/VIS_FPC_MULTI
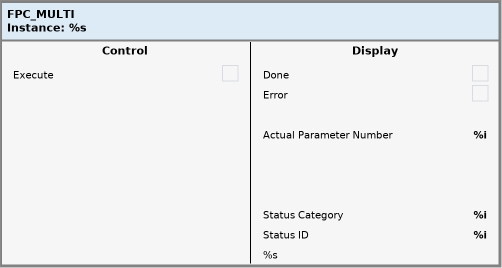
VISUALIZATION VIS_FPC_MULTI  // 502x268
VAR_INPUT
	{attribute 'parameterstringof' := 'm_Input_INST'}
	m_Input_INST_Str 	: STRING;
END_VAR
VAR_IN_OUT
	m_Input_INST 		: FPC_MULTI;
END_VAR
    Rectangle (0,1 500x265)
    Rectangle (0,1 500x40), "FPC_MULTI Instance: %s", text variable: m_Input_INST_Str
    Rectangle (260,245 240x20), "%s", text variable: m_Input_INST.Status.Msg
    Rectangle (430,125 60x20), "%i", text variable: m_Input_INST.ParamNo
    Label (10,65 120x20), "Execute"
    RoundedRectangle (222,65 16x16), colour toggle: m_Input_INST.Execute
        toggle m_Input_INST.Execute
    Label (260,65 120x20), "Done"
    Label (260,85 120x20), "Error"
    RoundedRectangle (472,65 16x16), colour toggle: m_Input_INST.Done
    RoundedRectangle (472,85 16x16), colour toggle: m_Input_INST.Error
    Label (260,125 140x20), "Actual Parameter Number"
    Label (0,41 250x20), "Control"
    Label (250,41 250x20), "Display"
    Line (250,42) (250,263)
    Rectangle (430,205 60x20), "%i", text variable: m_Input_INST.Status.Cat
    Label (260,205 128x20), "Status Category"
    Rectangle (430,225 60x20), "%i", text variable: m_Input_INST.Status.ID
    Label (260,225 128x20), "Status ID"
END_VISUALIZATION

// VISU/VIS_FPC_FILE_ARRAY
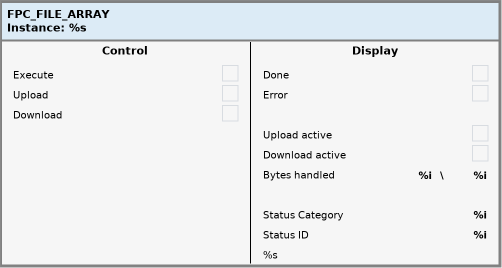
VISUALIZATION VIS_FPC_FILE_ARRAY  // 502x268
VAR_INPUT
	{attribute 'parameterstringof' := 'm_Input_INST'}
	m_Input_INST_Str 	: STRING;
END_VAR
VAR_IN_OUT
	m_Input_INST 		: FPC_FILE_ARRAY;
END_VAR
    Rectangle (0,1 500x265)
    Rectangle (0,1 500x40), "FPC_FILE_ARRAY Instance: %s", text variable: m_Input_INST_Str
    Rectangle (260,245 240x20), "%s", text variable: m_Input_INST.Status.Msg
    Label (10,65 120x20), "Execute"
    Label (10,85 120x20), "Upload"
    RoundedRectangle (222,65 16x16), colour toggle: m_Input_INST.Execute
        toggle m_Input_INST.Execute
    RoundedRectangle (222,85 16x16), colour toggle: m_Input_INST.Upload
        toggle m_Input_INST.Upload
    Label (260,65 120x20), "Done"
    Label (260,85 120x20), "Error"
    RoundedRectangle (472,65 16x16), colour toggle: m_Input_INST.Done
    RoundedRectangle (472,85 16x16), colour toggle: m_Input_INST.Error
    Label (0,41 250x20), "Control"
    Label (250,41 250x20), "Display"
    Line (250,42) (250,263)
    Rectangle (430,205 60x20), "%i", text variable: m_Input_INST.Status.Cat
    Label (260,205 128x20), "Status Category"
    Rectangle (430,225 60x20), "%i", text variable: m_Input_INST.Status.ID
    Label (260,225 128x20), "Status ID"
    Label (10,105 120x20), "Download"
    RoundedRectangle (222,105 16x16), colour toggle: m_Input_INST.Download
        toggle m_Input_INST.Download p2164770859=TRUE
    Rectangle (440,165 50x21), "%i", text variable: m_Input_INST.FileSize
    Label (260,125 120x20), "Upload active"
    Label (260,165 120x20), "Bytes handled"
    Label (260,145 120x20), "Download active"
    Rectangle (385,165 50x21), "%i", text variable: m_Input_INST.CountByte
    Label (437,165 13x21), "\"
    RoundedRectangle (472,125 16x16), colour toggle: m_Input_INST.vis_upload
    RoundedRectangle (472,145 16x16), colour toggle: m_Input_INST.vis_download
END_VISUALIZATION
